{attribute 'qualified_only'}
VAR_GLOBAL
	RpcBlock : FB_Rpc;
	
END_VAR

(* stored: Version 1.1.0.1, ProductVersion 3.1.4024.12
   GVL GVL_RPC: Id {000a9735-723b-4a0e-bba8-0261fd0b8c07} *)
